FUNCTION_BLOCK fbContext EXTENDS TcoCore.TcoContext
VAR
    {attribute addProperty Name "Toggle task example"}
    {attribute addProperty StateOnDesc "<#Enabled#>"}
    {attribute addProperty StateOffDesc "<#Disabled#>"}
    _toggleTaskExample : TcoCore.TcoToggleTask(THIS^, FALSE);
    {attribute addProperty Name "Momentary task example"}
    {attribute addProperty StateOnDesc "<#Running#>"}
    {attribute addProperty StateOffDesc "<#Stopped#>"}
    _momentaryTaskExample : TcoCore.TcoMomentaryTask(THIS^);
END_VAR

METHOD PROTECTED Main
_toggleTaskExample.Run();
_momentaryTaskExample.Run();
END_METHOD

END_FUNCTION_BLOCK

(* stored: Version 1.1.0.1
   POU fbContext: Id {2a1cec87-1ff7-064f-2678-b3fb1b407c7e}, SpecialFunc None
   Method Main: Id {17ff76c9-c8cb-0dc2-0912-164ab0c91c5e} *)
